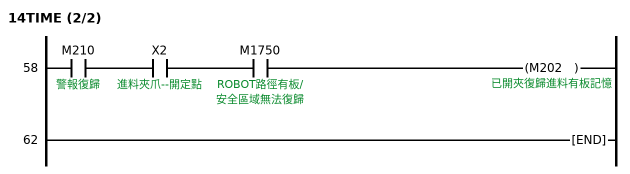
[picture p72: ladder of 14TIME, rungs at steps 58 to 62]
58    LD      M210  ; 警報復歸
      AND     X2  ; 進料夾爪--開定點
      AND     M1750  ; ROBOT路徑有板/安全區域無法復歸
      OUT     M202  ; 已開夾復歸進料有板記憶
62    END
END_PROGRAM

PROGRAM 15STATUS
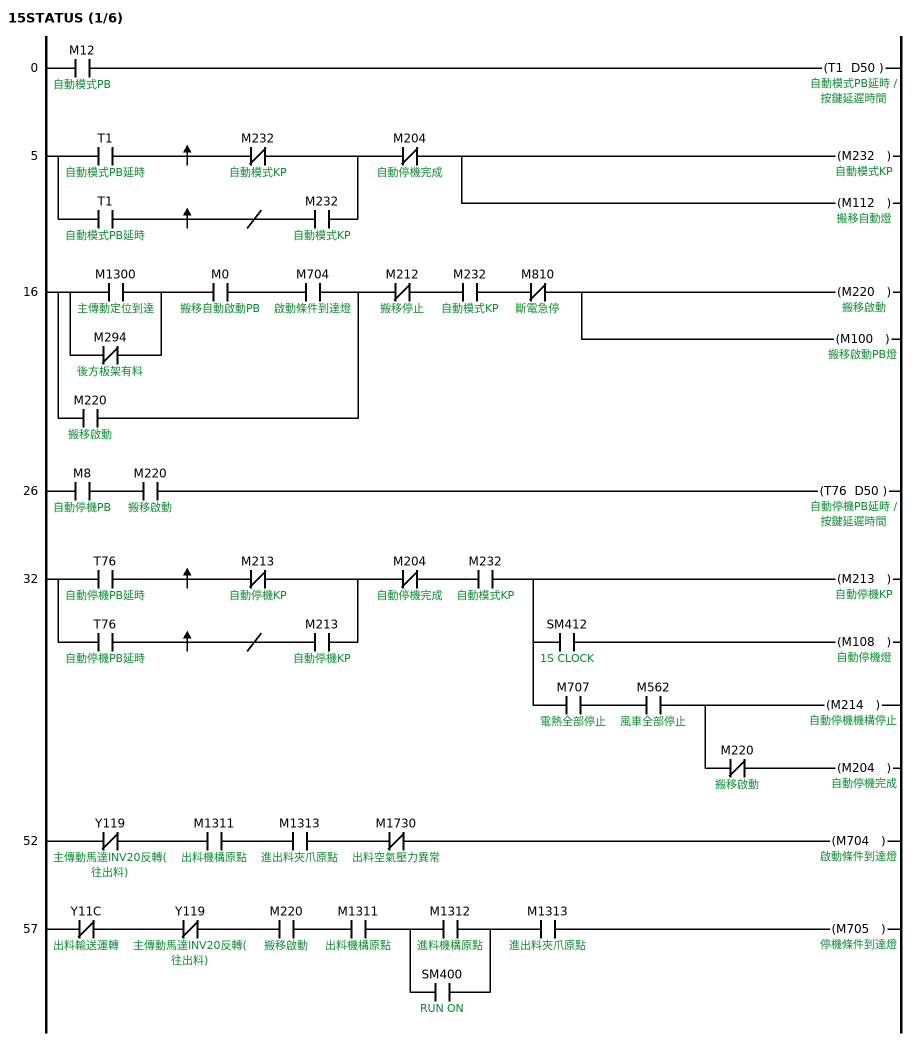
0     LD      M12  ; 自動模式PB
      OUT     T1 D50  ; 自動模式PB延時 / 按鍵延遲時間
5     LD      T1  ; 自動模式PB延時
      MEP
      ANI     M232  ; 自動模式KP
      LD      T1  ; 自動模式PB延時
      MEP
      INV
      AND     M232  ; 自動模式KP
      ORB
      ANI     M204  ; 自動停機完成
      OUT     M232  ; 自動模式KP
      OUT     M112  ; 搬移自動燈
16    LD      M1300  ; 主傳動定位到達
      ORI     M294  ; 後方板架有料
      AND     M0  ; 搬移自動啟動PB
      AND     M704  ; 啟動條件到達燈
      OR      M220  ; 搬移啟動
      ANI     M212  ; 搬移停止
      AND     M232  ; 自動模式KP
      ANI     M810  ; 斷電急停
      OUT     M220  ; 搬移啟動
      OUT     M100  ; 搬移啟動PB燈
26    LD      M8  ; 自動停機PB
      AND     M220  ; 搬移啟動
      OUT     T76 D50  ; 自動停機PB延時 / 按鍵延遲時間
32    LD      T76  ; 自動停機PB延時
      MEP
      ANI     M213  ; 自動停機KP
      LD      T76  ; 自動停機PB延時
      MEP
      INV
      AND     M213  ; 自動停機KP
      ORB
      ANI     M204  ; 自動停機完成
      AND     M232  ; 自動模式KP
      OUT     M213  ; 自動停機KP
      MPS
      AND     SM412  ; 1S CLOCK
      OUT     M108  ; 自動停機燈
      MPP
      AND     M707  ; 電熱全部停止
      AND     M562  ; 風車全部停止
      OUT     M214  ; 自動停機機構停止
      ANI     M220  ; 搬移啟動
      OUT     M204  ; 自動停機完成
52    LDI     Y119  ; 主傳動馬達INV20反轉(往出料)
      AND     M1311  ; 出料機構原點
      AND     M1313  ; 進出料夾爪原點
      ANI     M1730  ; 出料空氣壓力異常
      OUT     M704  ; 啟動條件到達燈
57    LDI     Y11C  ; 出料輸送運轉
      ANI     Y119  ; 主傳動馬達INV20反轉(往出料)
      AND     M220  ; 搬移啟動
      AND     M1311  ; 出料機構原點
      LD      M1312  ; 進料機構原點
      OR      SM400  ; RUN ON
      ANB
      AND     M1313  ; 進出料夾爪原點
      OUT     M705  ; 停機條件到達燈
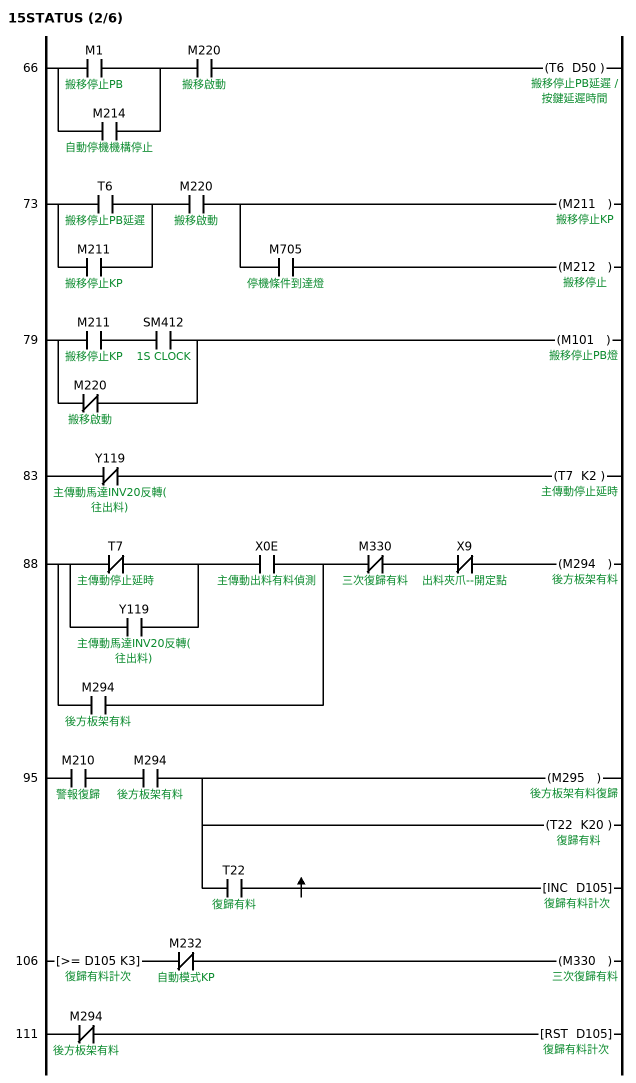
66    LD      M1  ; 搬移停止PB
      OR      M214  ; 自動停機機構停止
      AND     M220  ; 搬移啟動
      OUT     T6 D50  ; 搬移停止PB延遲 / 按鍵延遲時間
73    LD      T6  ; 搬移停止PB延遲
      OR      M211  ; 搬移停止KP
      AND     M220  ; 搬移啟動
      OUT     M211  ; 搬移停止KP
      AND     M705  ; 停機條件到達燈
      OUT     M212  ; 搬移停止
79    LD      M211  ; 搬移停止KP
      AND     SM412  ; 1S CLOCK
      ORI     M220  ; 搬移啟動
      OUT     M101  ; 搬移停止PB燈
83    LDI     Y119  ; 主傳動馬達INV20反轉(往出料)
      OUT     T7 K2  ; 主傳動停止延時
88    LDI     T7  ; 主傳動停止延時
      OR      Y119  ; 主傳動馬達INV20反轉(往出料)
      AND     X0E  ; 主傳動出料有料偵測
      OR      M294  ; 後方板架有料
      ANI     M330  ; 三次復歸有料
      ANI     X9  ; 出料夾爪--開定點
      OUT     M294  ; 後方板架有料
95    LD      M210  ; 警報復歸
      AND     M294  ; 後方板架有料
      OUT     M295  ; 後方板架有料復歸
      OUT     T22 K20  ; 復歸有料
      AND     T22  ; 復歸有料
      MEP
      INC     D105  ; 復歸有料計次
106   LD>=    D105 K3  ; 復歸有料計次
      ANI     M232  ; 自動模式KP
      OUT     M330  ; 三次復歸有料
111   LDI     M294  ; 後方板架有料
      RST     D105  ; 復歸有料計次
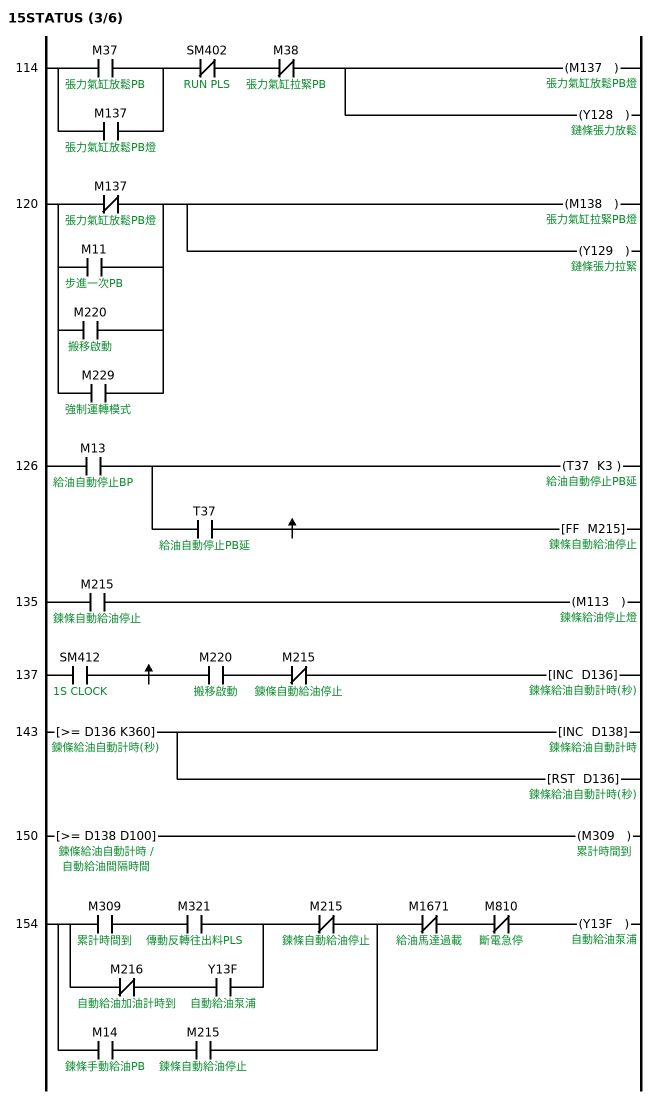
114   LD      M37  ; 張力氣缸放鬆PB
      OR      M137  ; 張力氣缸放鬆PB燈
      ANI     SM402  ; RUN PLS
      ANI     M38  ; 張力氣缸拉緊PB
      OUT     M137  ; 張力氣缸放鬆PB燈
      OUT     Y128  ; 鏈條張力放鬆
120   LDI     M137  ; 張力氣缸放鬆PB燈
      OR      M11  ; 步進一次PB
      OR      M220  ; 搬移啟動
      OR      M229  ; 強制運轉模式
      OUT     M138  ; 張力氣缸拉緊PB燈
      OUT     Y129  ; 鏈條張力拉緊
126   LD      M13  ; 給油自動停止BP
      OUT     T37 K3  ; 給油自動停止PB延
      AND     T37  ; 給油自動停止PB延
      MEP
      FF      M215  ; 鍊條自動給油停止
135   LD      M215  ; 鍊條自動給油停止
      OUT     M113  ; 鍊條給油停止燈
137   LD      SM412  ; 1S CLOCK
      MEP
      AND     M220  ; 搬移啟動
      ANI     M215  ; 鍊條自動給油停止
      INC     D136  ; 鍊條給油自動計時(秒)
143   LD>=    D136 K360  ; 鍊條給油自動計時(秒)
      INC     D138  ; 鍊條給油自動計時
      RST     D136  ; 鍊條給油自動計時(秒)
150   LD>=    D138 D100  ; 鍊條給油自動計時 / 自動給油間隔時間
      OUT     M309  ; 累計時間到
154   LD      M309  ; 累計時間到
      AND     M321  ; 傳動反轉往出料PLS
      LDI     M216  ; 自動給油加油計時到
      AND     Y13F  ; 自動給油泵浦
      ORB
      ANI     M215  ; 鍊條自動給油停止
      LD      M14  ; 鍊條手動給油PB
      AND     M215  ; 鍊條自動給油停止
      ORB
      ANI     M1671  ; 給油馬達過載
      ANI     M810  ; 斷電急停
      OUT     Y13F  ; 自動給油泵浦
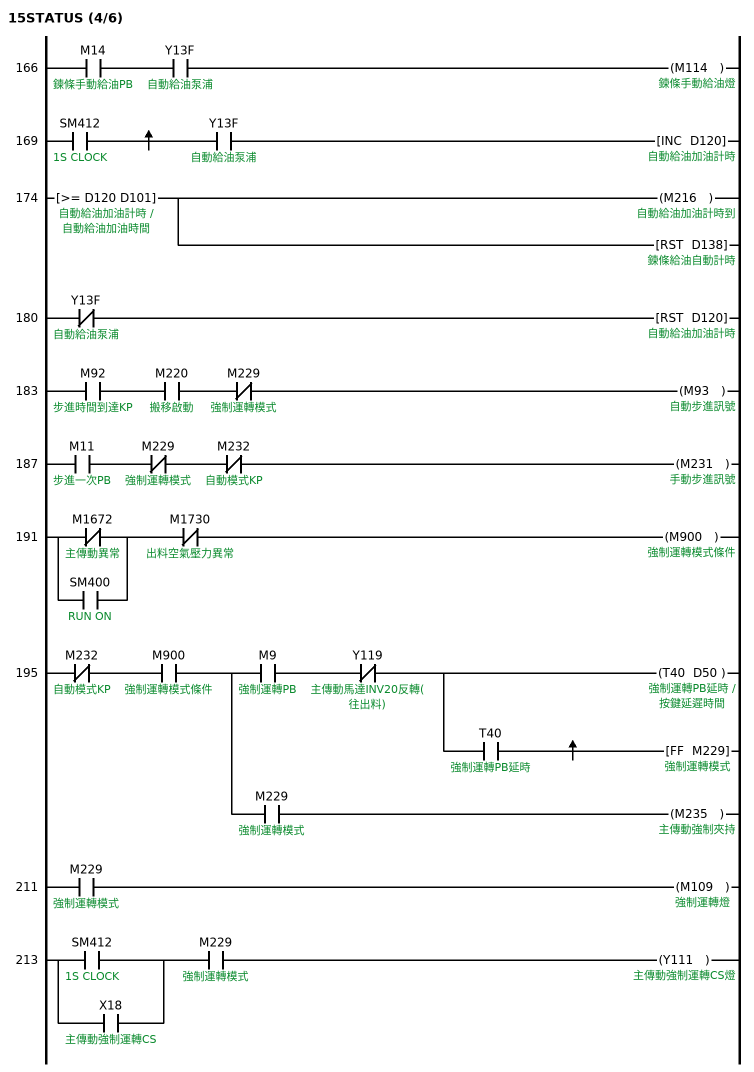
166   LD      M14  ; 鍊條手動給油PB
      AND     Y13F  ; 自動給油泵浦
      OUT     M114  ; 鍊條手動給油燈
169   LD      SM412  ; 1S CLOCK
      MEP
      AND     Y13F  ; 自動給油泵浦
      INC     D120  ; 自動給油加油計時
174   LD>=    D120 D101  ; 自動給油加油計時 / 自動給油加油時間
      OUT     M216  ; 自動給油加油計時到
      RST     D138  ; 鍊條給油自動計時
180   LDI     Y13F  ; 自動給油泵浦
      RST     D120  ; 自動給油加油計時
183   LD      M92  ; 步進時間到達KP
      AND     M220  ; 搬移啟動
      ANI     M229  ; 強制運轉模式
      OUT     M93  ; 自動步進訊號
187   LD      M11  ; 步進一次PB
      ANI     M229  ; 強制運轉模式
      ANI     M232  ; 自動模式KP
      OUT     M231  ; 手動步進訊號
191   LDI     M1672  ; 主傳動異常
      OR      SM400  ; RUN ON
      ANI     M1730  ; 出料空氣壓力異常
      OUT     M900  ; 強制運轉模式條件
195   LDI     M232  ; 自動模式KP
      AND     M900  ; 強制運轉模式條件
      MPS
      AND     M9  ; 強制運轉PB
      ANI     Y119  ; 主傳動馬達INV20反轉(往出料)
      OUT     T40 D50  ; 強制運轉PB延時 / 按鍵延遲時間
      AND     T40  ; 強制運轉PB延時
      MEP
      FF      M229
      MPP
      AND     M229  ; 強制運轉模式
      OUT     M235  ; 主傳動強制夾持
211   LD      M229  ; 強制運轉模式
      OUT     M109  ; 強制運轉燈
213   LD      SM412  ; 1S CLOCK
      OR      X18  ; 主傳動強制運轉CS
      AND     M229  ; 強制運轉模式
      OUT     Y111  ; 主傳動強制運轉CS燈
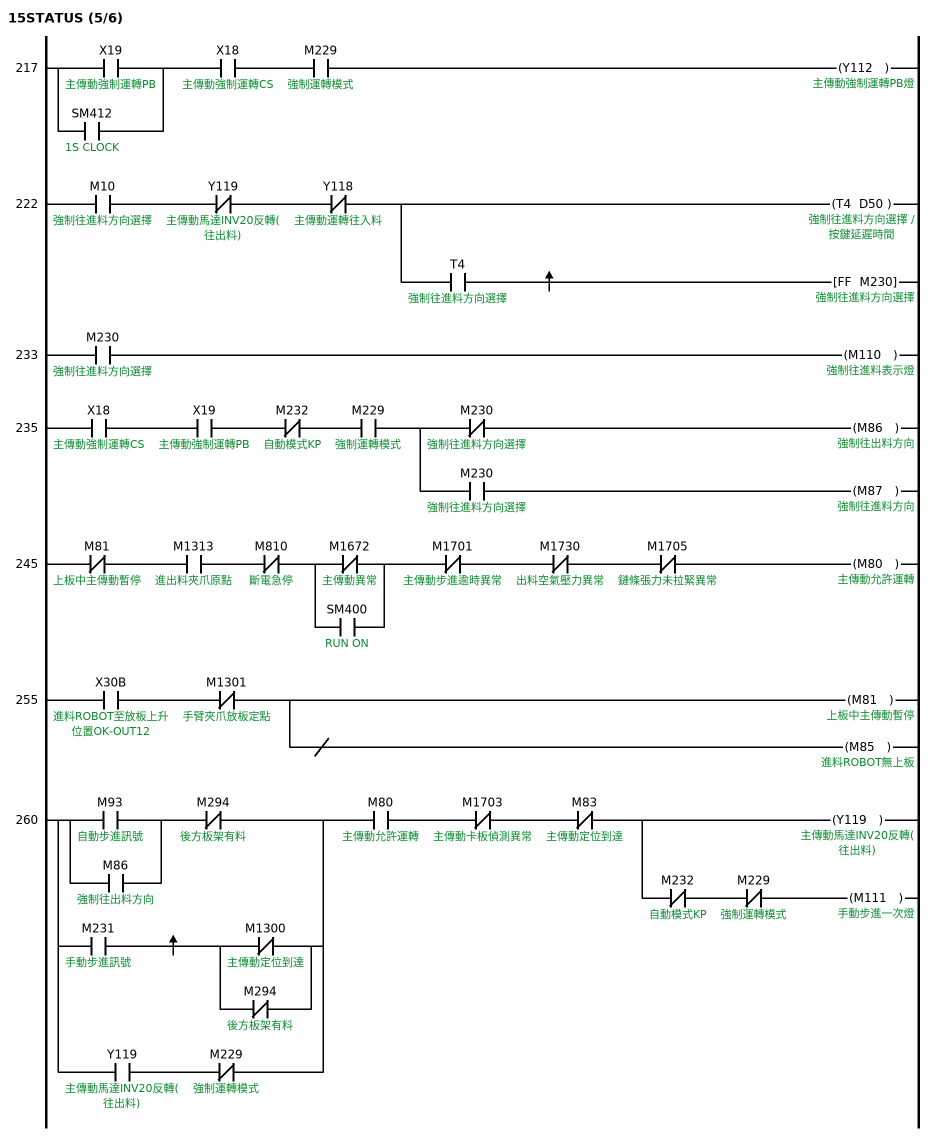
217   LD      X19  ; 主傳動強制運轉PB
      OR      SM412  ; 1S CLOCK
      AND     X18  ; 主傳動強制運轉CS
      AND     M229  ; 強制運轉模式
      OUT     Y112  ; 主傳動強制運轉PB燈
222   LD      M10  ; 強制往進料方向選擇
      ANI     Y119  ; 主傳動馬達INV20反轉(往出料)
      ANI     Y118  ; 主傳動運轉往入料
      OUT     T4 D50  ; 強制往進料方向選擇 / 按鍵延遲時間
      AND     T4  ; 強制往進料方向選擇
      MEP
      FF      M230  ; 強制往進料方向選擇
233   LD      M230  ; 強制往進料方向選擇
      OUT     M110  ; 強制往進料表示燈
235   LD      X18  ; 主傳動強制運轉CS
      AND     X19  ; 主傳動強制運轉PB
      ANI     M232  ; 自動模式KP
      AND     M229  ; 強制運轉模式
      MPS
      ANI     M230  ; 強制往進料方向選擇
      OUT     M86  ; 強制往出料方向
      MPP
      AND     M230  ; 強制往進料方向選擇
      OUT     M87  ; 強制往進料方向
245   LDI     M81  ; 上板中主傳動暫停
      AND     M1313  ; 進出料夾爪原點
      ANI     M810  ; 斷電急停
      LDI     M1672  ; 主傳動異常
      OR      SM400  ; RUN ON
      ANB
      ANI     M1701  ; 主傳動步進逾時異常
      ANI     M1730  ; 出料空氣壓力異常
      ANI     M1705  ; 鏈條張力未拉緊異常
      OUT     M80  ; 主傳動允許運轉
255   LD      X30B  ; 進料ROBOT至放板上升位置OK-OUT12
      ANI     M1301  ; 手臂夾爪放板定點
      OUT     M81  ; 上板中主傳動暫停
      INV
      OUT     M85  ; 進料ROBOT無上板
260   LD      M93  ; 自動步進訊號
      OR      M86  ; 強制往出料方向
      ANI     M294  ; 後方板架有料
      LD      M231  ; 手動步進訊號
      MEP
      LDI     M1300  ; 主傳動定位到達
      ORI     M294  ; 後方板架有料
      ANB
      ORB
      LD      Y119  ; 主傳動馬達INV20反轉(往出料)
      ANI     M229  ; 強制運轉模式
      ORB
      AND     M80  ; 主傳動允許運轉
      ANI     M1703  ; 主傳動卡板偵測異常
      ANI     M83  ; 主傳動定位到達
      OUT     Y119  ; 主傳動馬達INV20反轉(往出料)
      ANI     M232  ; 自動模式KP
      ANI     M229  ; 強制運轉模式
      OUT     M111  ; 手動步進一次燈
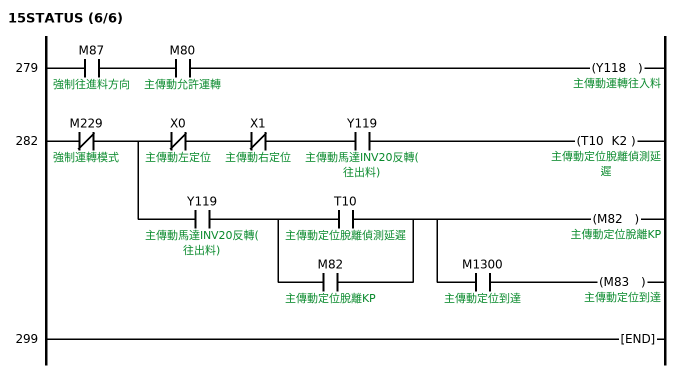
279   LD      M87  ; 強制往進料方向
      AND     M80  ; 主傳動允許運轉
      OUT     Y118  ; 主傳動運轉往入料
282   LDI     M229  ; 強制運轉模式
      MPS
      ANI     X0  ; 主傳動左定位
      ANI     X1  ; 主傳動右定位
      AND     Y119  ; 主傳動馬達INV20反轉(往出料)
      OUT     T10 K2  ; 主傳動定位脫離偵測延遲
      MPP
      AND     Y119  ; 主傳動馬達INV20反轉(往出料)
      LD      T10  ; 主傳動定位脫離偵測延遲
      OR      M82  ; 主傳動定位脫離KP
      ANB
      OUT     M82  ; 主傳動定位脫離KP
      AND     M1300  ; 主傳動定位到達
      OUT     M83  ; 主傳動定位到達
299   END
END_PROGRAM

PROGRAM 21SECS
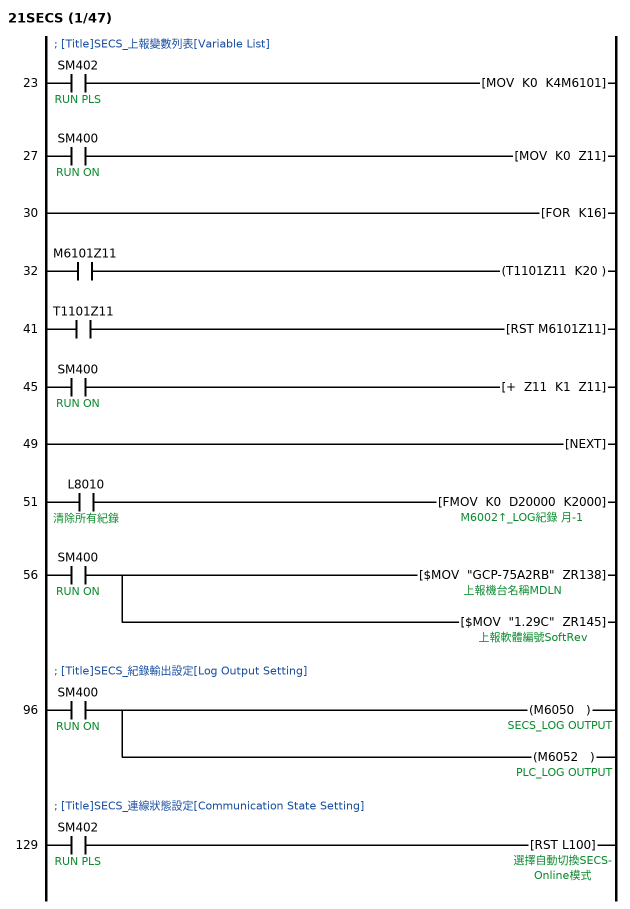
; [Title]SECS_上報變數列表[Variable List]
23    LD      SM402  ; RUN PLS
      MOV     K0 K4M6101  ; EQP->SES控制模式切換(Online/Off)
27    LD      SM400  ; RUN ON
      MOV     K0 Z11
30    FOR     K16
32    LD      M6101Z11
      OUT     T1101Z11 K20
41    LD      T1101Z11
      RST     M6101Z11
45    LD      SM400  ; RUN ON
      +       Z11 K1 Z11
49    NEXT
51    LD      L8010  ; 清除所有紀錄
      FMOV    K0 D20000 K2000  ; M6002↑_LOG紀錄 月-1
56    LD      SM400  ; RUN ON
      $MOV    "GCP-75A2RB" ZR138  ; 上報機台名稱MDLN
      $MOV    "1.29C" ZR145  ; 上報軟體編號SoftRev
; [Title]SECS_紀錄輸出設定[Log Output Setting]
96    LD      SM400  ; RUN ON
      OUT     M6050  ; SECS_LOG OUTPUT
      OUT     M6052  ; PLC_LOG OUTPUT
; [Title]SECS_連線狀態設定[Communication State Setting]
129   LD      SM402  ; RUN PLS
      RST     L100  ; 選擇自動切換SECS-Online模式
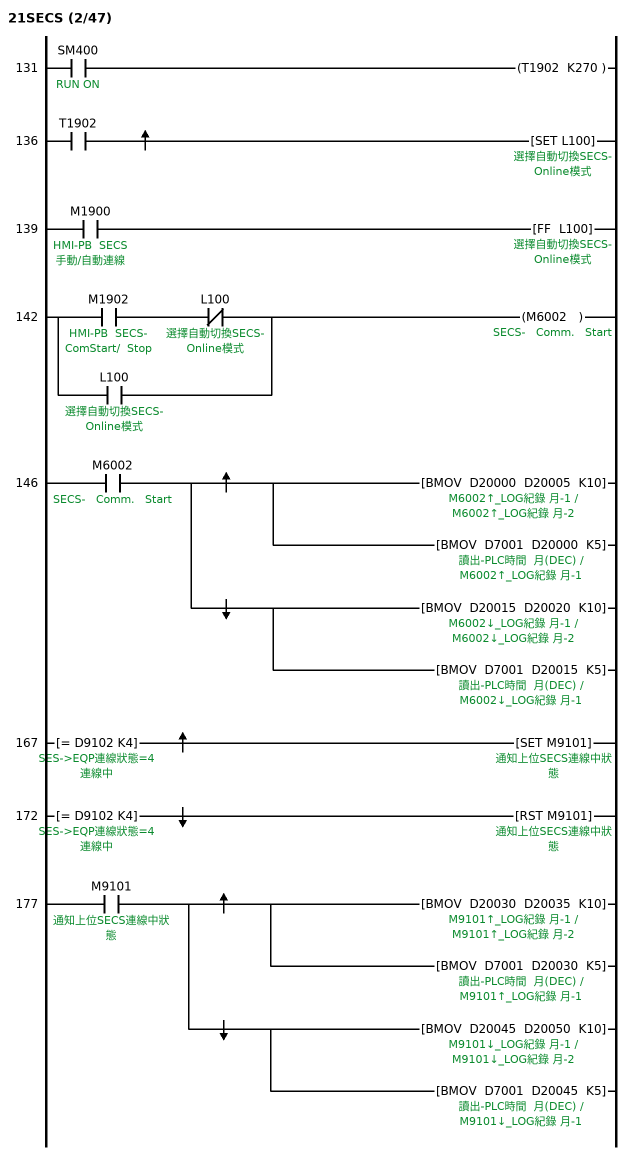
131   LD      SM400  ; RUN ON
      OUT     T1902 K270
136   LD      T1902
      MEP
      SET     L100  ; 選擇自動切換SECS-Online模式
139   LD      M1900  ; HMI-PB  SECS    手動/自動連線
      FF      L100
142   LD      M1902  ; HMI-PB  SECS-ComStart/  Stop
      ANI     L100  ; 選擇自動切換SECS-Online模式
      OR      L100  ; 選擇自動切換SECS-Online模式
      OUT     M6002  ; SECS-   Comm.   Start
146   LD      M6002  ; SECS-   Comm.   Start
      MPS
      MEP
      BMOV    D20000 D20005 K10  ; M6002↑_LOG紀錄 月-2
      BMOV    D7001 D20000 K5  ; 讀出-PLC時間  月(DEC)
      MPP
      MEF
      BMOV    D20015 D20020 K10  ; M6002↓_LOG紀錄 月-1 / M6002↓_LOG紀錄 月-2
      BMOV    D7001 D20015 K5
167   LD=     D9102 K4  ; SES->EQP連線狀態=4      連線中
      MEP
      SET     M9101  ; 通知上位SECS連線中狀態
172   LD=     D9102 K4  ; SES->EQP連線狀態=4      連線中
      MEF
      RST     M9101  ; 通知上位SECS連線中狀態
177   LD      M9101  ; 通知上位SECS連線中狀態
      MPS
      MEP
      BMOV    D20030 D20035 K10  ; M9101↑_LOG紀錄 月-1 / M9101↑_LOG紀錄 月-2
      BMOV    D7001 D20030 K5
      MPP
      MEF
      BMOV    D20045 D20050 K10  ; M9101↓_LOG紀錄 月-1 / M9101↓_LOG紀錄 月-2
      BMOV    D7001 D20045 K5
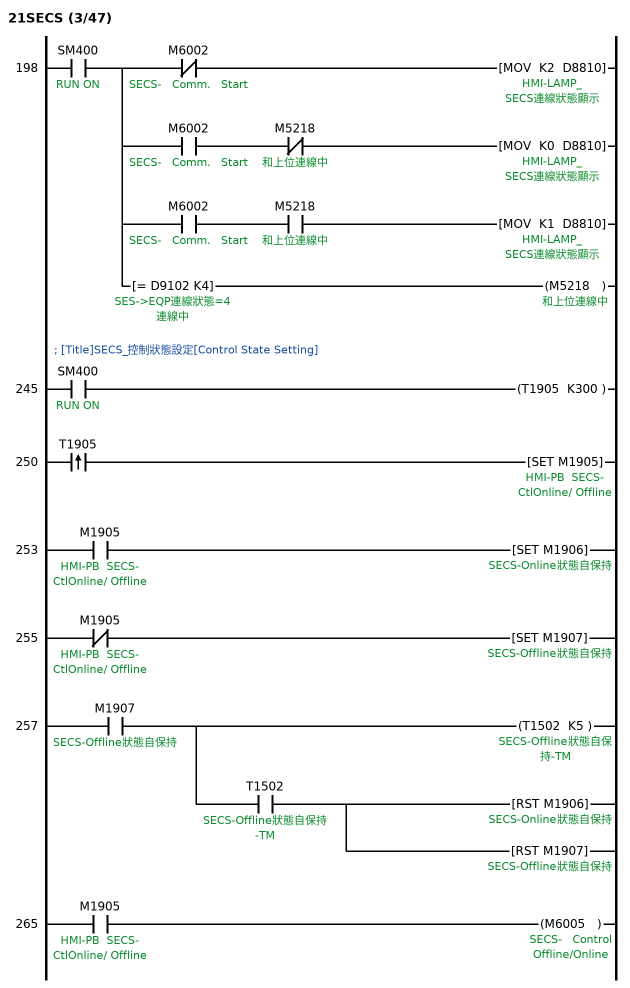
198   LD      SM400  ; RUN ON
      MPS
      ANI     M6002  ; SECS-   Comm.   Start
      MOV     K2 D8810  ; HMI-LAMP_SECS連線狀態顯示
      MRD
      AND     M6002  ; SECS-   Comm.   Start
      ANI     M5218  ; 和上位連線中
      MOV     K0 D8810
      MRD
      AND     M6002  ; SECS-   Comm.   Start
      AND     M5218  ; 和上位連線中
      MOV     K1 D8810
      MPP
      AND=    D9102 K4  ; SES->EQP連線狀態=4      連線中
      OUT     M5218  ; 和上位連線中
; [Title]SECS_控制狀態設定[Control State Setting]
245   LD      SM400  ; RUN ON
      OUT     T1905 K300
250   LDP     T1905
      SET     M1905  ; HMI-PB  SECS-CtlOnline/ Offline
253   LD      M1905  ; HMI-PB  SECS-CtlOnline/ Offline
      SET     M1906  ; SECS-Online狀態自保持
255   LDI     M1905  ; HMI-PB  SECS-CtlOnline/ Offline
      SET     M1907  ; SECS-Offline狀態自保持
257   LD      M1907  ; SECS-Offline狀態自保持
      OUT     T1502 K5  ; SECS-Offline狀態自保持-TM
      AND     T1502  ; SECS-Offline狀態自保持-TM
      RST     M1906  ; SECS-Online狀態自保持
      RST     M1907  ; SECS-Offline狀態自保持
265   LD      M1905  ; HMI-PB  SECS-CtlOnline/ Offline
      OUT     M6005  ; SECS-   Control Offline/Online
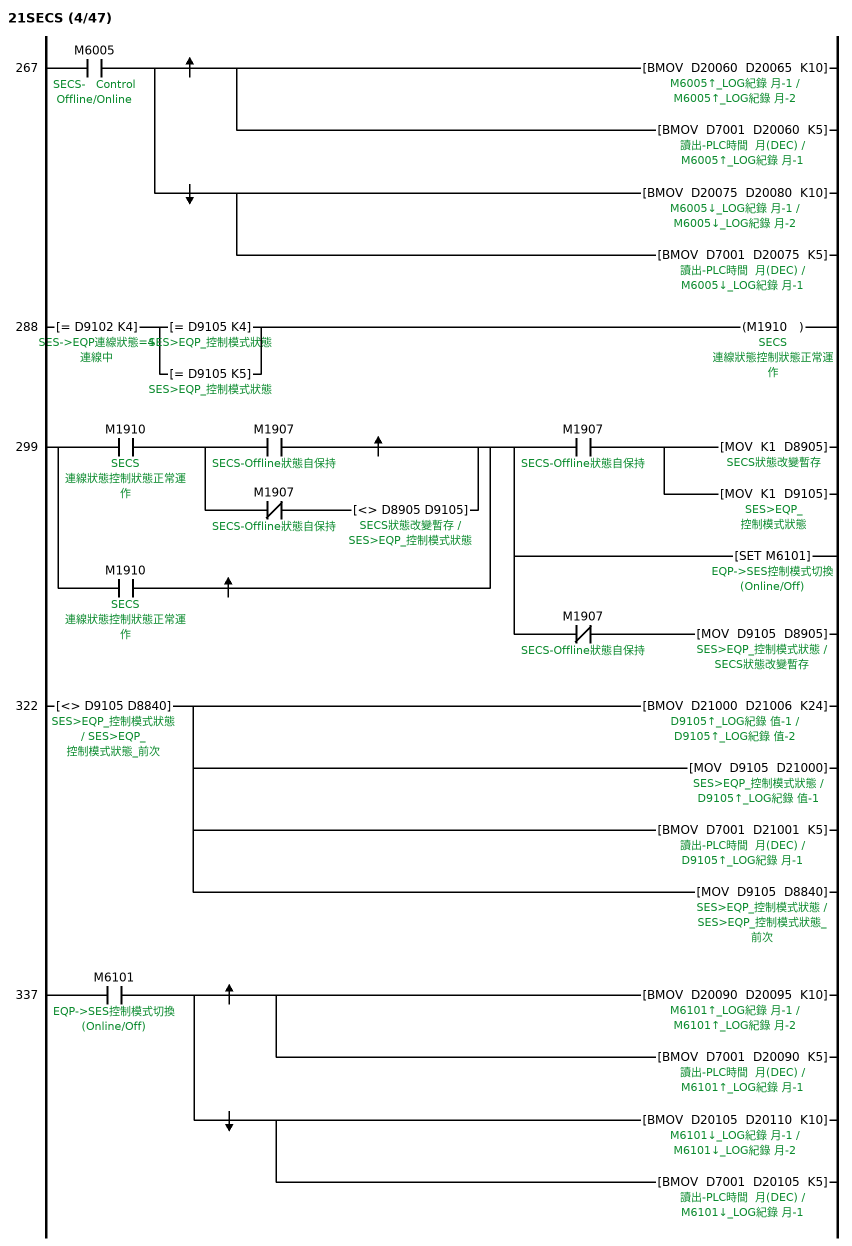
267   LD      M6005  ; SECS-   Control Offline/Online
      MPS
      MEP
      BMOV    D20060 D20065 K10  ; M6005↑_LOG紀錄 月-1 / M6005↑_LOG紀錄 月-2
      BMOV    D7001 D20060 K5
      MPP
      MEF
      BMOV    D20075 D20080 K10  ; M6005↓_LOG紀錄 月-1 / M6005↓_LOG紀錄 月-2
      BMOV    D7001 D20075 K5
288   LD=     D9102 K4  ; SES->EQP連線狀態=4      連線中
      LD=     D9105 K4  ; SES>EQP_控制模式狀態
      OR=     D9105 K5  ; SES>EQP_控制模式狀態
      ANB
      OUT     M1910  ; SECS    連線狀態控制狀態正常運作
299   LD      M1910  ; SECS    連線狀態控制狀態正常運作
      LD      M1907  ; SECS-Offline狀態自保持
      MEP
      LDI     M1907  ; SECS-Offline狀態自保持
      AND<>   D8905 D9105  ; SECS狀態改變暫存 / SES>EQP_控制模式狀態
      ORB
      ANB
      LD      M1910  ; SECS    連線狀態控制狀態正常運作
      MEP
      ORB
      MPS
      AND     M1907  ; SECS-Offline狀態自保持
      MOV     K1 D8905
      MOV     K1 D9105
      MPP
      SET     M6101  ; EQP->SES控制模式切換(Online/Off)
      ANI     M1907  ; SECS-Offline狀態自保持
      MOV     D9105 D8905
322   LD<>    D9105 D8840  ; SES>EQP_控制模式狀態 / SES>EQP_控制模式狀態_前次
      BMOV    D21000 D21006 K24  ; D9105↑_LOG紀錄 值-1 / D9105↑_LOG紀錄 值-2
      MOV     D9105 D21000
      BMOV    D7001 D21001 K5  ; D9105↑_LOG紀錄 月-1
      MOV     D9105 D8840
337   LD      M6101  ; EQP->SES控制模式切換(Online/Off)
      MPS
      MEP
      BMOV    D20090 D20095 K10  ; M6101↑_LOG紀錄 月-1 / M6101↑_LOG紀錄 月-2
      BMOV    D7001 D20090 K5
      MPP
      MEF
      BMOV    D20105 D20110 K10  ; M6101↓_LOG紀錄 月-1 / M6101↓_LOG紀錄 月-2
      BMOV    D7001 D20105 K5
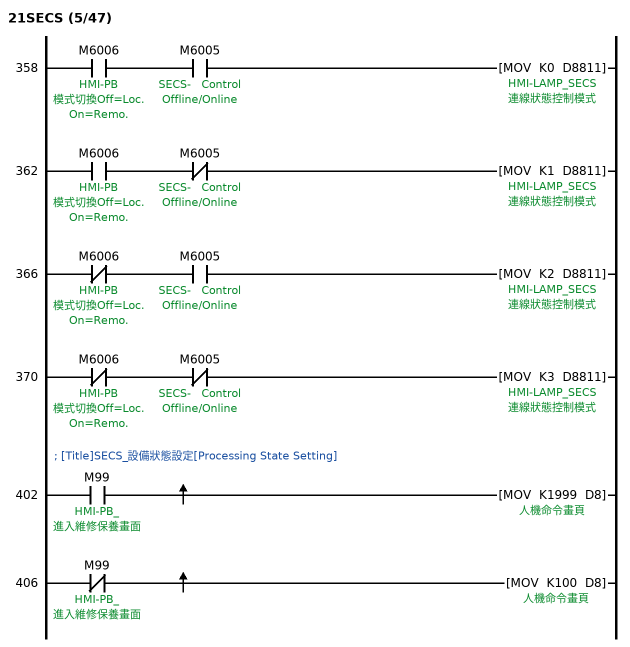
358   LD      M6006  ; HMI-PB  模式切換Off=Loc.On=Remo.
      AND     M6005  ; SECS-   Control Offline/Online
      MOV     K0 D8811  ; HMI-LAMP_SECS   連線狀態控制模式
362   LD      M6006  ; HMI-PB  模式切換Off=Loc.On=Remo.
      ANI     M6005  ; SECS-   Control Offline/Online
      MOV     K1 D8811
366   LDI     M6006  ; HMI-PB  模式切換Off=Loc.On=Remo.
      AND     M6005  ; SECS-   Control Offline/Online
      MOV     K2 D8811
370   LDI     M6006  ; HMI-PB  模式切換Off=Loc.On=Remo.
      ANI     M6005  ; SECS-   Control Offline/Online
      MOV     K3 D8811
; [Title]SECS_設備狀態設定[Processing State Setting]
402   LD      M99  ; HMI-PB_ 進入維修保養畫面
      MEP
      MOV     K1999 D8  ; 人機命令畫頁
406   LDI     M99  ; HMI-PB_ 進入維修保養畫面
      MEP
      MOV     K100 D8
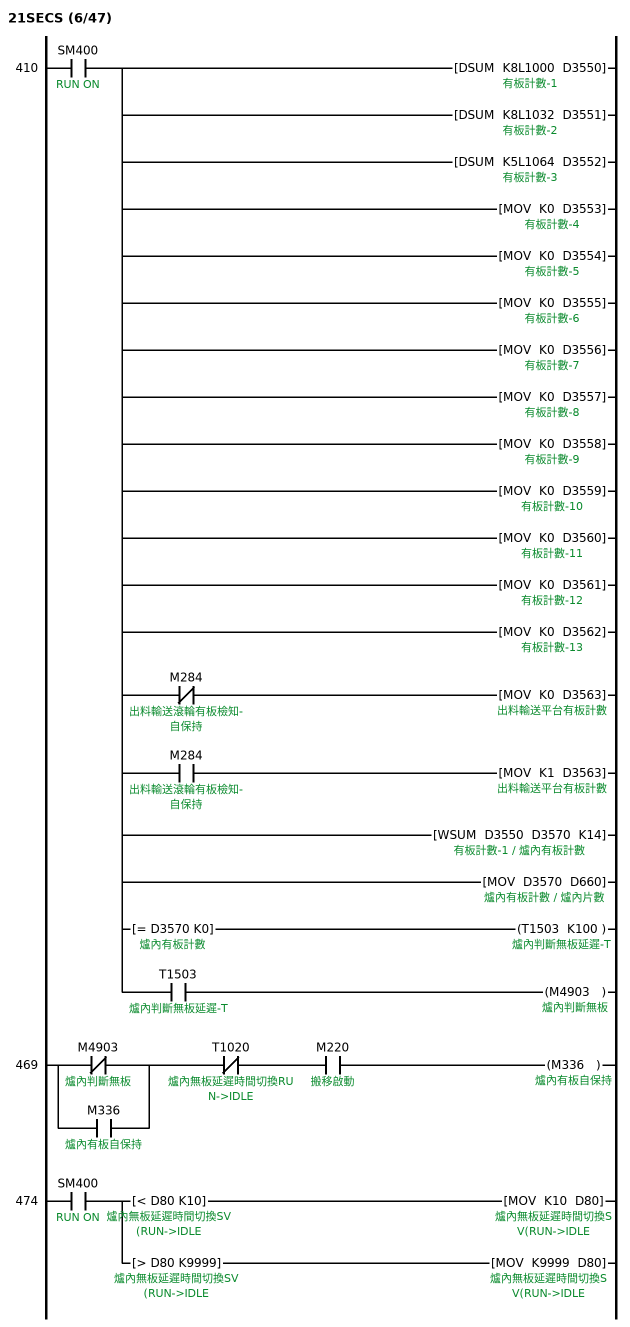
410   LD      SM400  ; RUN ON
      DSUM    K8L1000 D3550  ; 上板記憶 / 有板計數-1
      DSUM    K8L1032 D3551  ; 上板記憶 / 有板計數-2
      DSUM    K5L1064 D3552  ; 上板記憶 / 有板計數-3
      MOV     K0 D3553  ; 有板計數-4
      MOV     K0 D3554  ; 有板計數-5
      MOV     K0 D3555  ; 有板計數-6
      MOV     K0 D3556  ; 有板計數-7
      MOV     K0 D3557  ; 有板計數-8
      MOV     K0 D3558  ; 有板計數-9
      MOV     K0 D3559  ; 有板計數-10
      MOV     K0 D3560  ; 有板計數-11
      MOV     K0 D3561  ; 有板計數-12
      MOV     K0 D3562  ; 有板計數-13
      MPS
      ANI     M284  ; 出料輸送滾輪有板檢知-自保持
      MOV     K0 D3563  ; 出料輸送平台有板計數
      MRD
      AND     M284  ; 出料輸送滾輪有板檢知-自保持
      MOV     K1 D3563
      MPP
      WSUM    D3550 D3570 K14  ; 爐內有板計數
      MOV     D3570 D660  ; 爐內片數
      MPS
      AND=    D3570 K0  ; 爐內有板計數
      OUT     T1503 K100  ; 爐內判斷無板延遲-T
      MPP
      AND     T1503  ; 爐內判斷無板延遲-T
      OUT     M4903  ; 爐內判斷無板
469   LDI     M4903  ; 爐內判斷無板
      OR      M336  ; 爐內有板自保持
      ANI     T1020  ; 爐內無板延遲時間切換RUN->IDLE
      AND     M220  ; 搬移啟動
      OUT     M336  ; 爐內有板自保持
474   LD      SM400  ; RUN ON
      MPS
      AND<    D80 K10  ; 爐內無板延遲時間切換SV(RUN->IDLE
      MOV     K10 D80
      MPP
      AND>    D80 K9999  ; 爐內無板延遲時間切換SV(RUN->IDLE
      MOV     K9999 D80
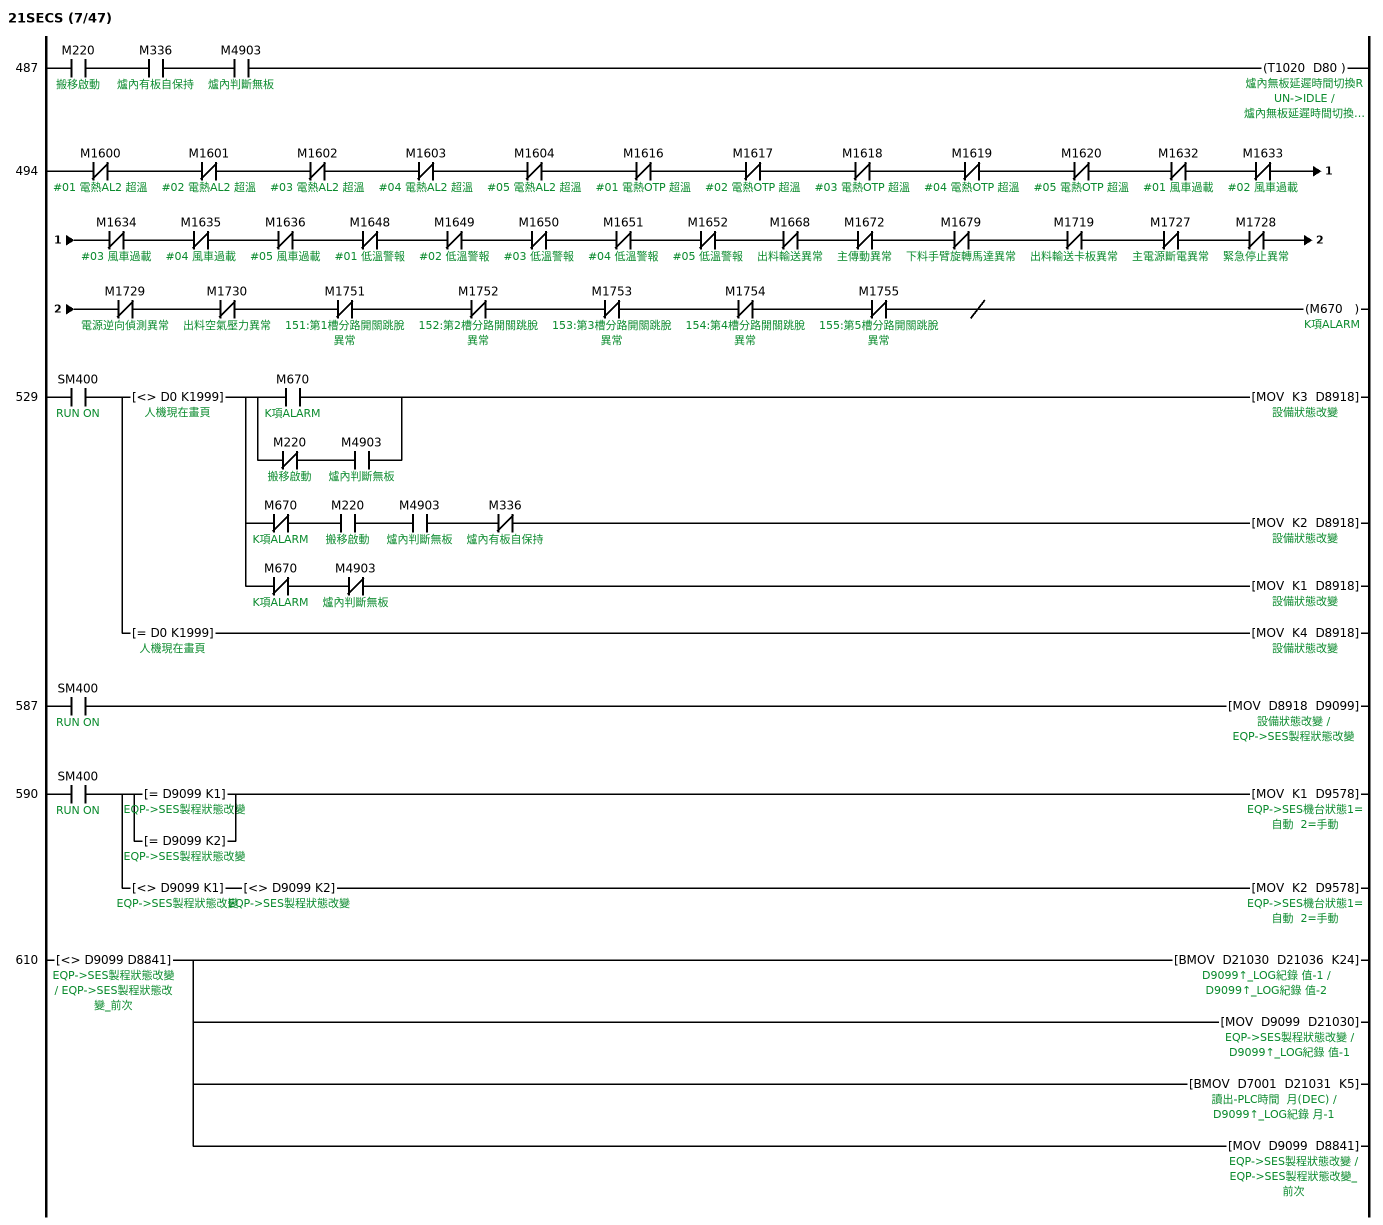
487   LD      M220  ; 搬移啟動
      AND     M336  ; 爐內有板自保持
      AND     M4903  ; 爐內判斷無板
      OUT     T1020 D80  ; 爐內無板延遲時間切換RUN->IDLE / 爐內無板延遲時間切換SV(RUN->IDLE
494   LDI     M1600  ; #01 電熱AL2 超溫
      ANI     M1601  ; #02 電熱AL2 超溫
      ANI     M1602  ; #03 電熱AL2 超溫
      ANI     M1603  ; #04 電熱AL2 超溫
      ANI     M1604  ; #05 電熱AL2 超溫
      ANI     M1616  ; #01 電熱OTP 超溫
      ANI     M1617  ; #02 電熱OTP 超溫
      ANI     M1618  ; #03 電熱OTP 超溫
      ANI     M1619  ; #04 電熱OTP 超溫
      ANI     M1620  ; #05 電熱OTP 超溫
      ANI     M1632  ; #01 風車過載
      ANI     M1633  ; #02 風車過載
      ANI     M1634  ; #03 風車過載
      ANI     M1635  ; #04 風車過載
      ANI     M1636  ; #05 風車過載
      ANI     M1648  ; #01 低溫警報
      ANI     M1649  ; #02 低溫警報
      ANI     M1650  ; #03 低溫警報
      ANI     M1651  ; #04 低溫警報
      ANI     M1652  ; #05 低溫警報
      ANI     M1668  ; 出料輸送異常
      ANI     M1672  ; 主傳動異常
      ANI     M1679  ; 下料手臂旋轉馬達異常
      ANI     M1719  ; 出料輸送卡板異常
      ANI     M1727  ; 主電源斷電異常
      ANI     M1728  ; 緊急停止異常
      ANI     M1729  ; 電源逆向偵測異常
      ANI     M1730  ; 出料空氣壓力異常
      ANI     M1751  ; 151:第1槽分路開關跳脫異常
      ANI     M1752  ; 152:第2槽分路開關跳脫異常
      ANI     M1753  ; 153:第3槽分路開關跳脫異常
      ANI     M1754  ; 154:第4槽分路開關跳脫異常
      ANI     M1755  ; 155:第5槽分路開關跳脫異常
      INV
      OUT     M670  ; K項ALARM
529   LD      SM400  ; RUN ON
      MPS
      AND<>   D0 K1999  ; 人機現在畫頁
      MPS
      LD      M670  ; K項ALARM
      LDI     M220  ; 搬移啟動
      AND     M4903  ; 爐內判斷無板
      ORB
      ANB
      MOV     K3 D8918  ; 設備狀態改變
        [note] State=DOWN
      MRD
      ANI     M670  ; K項ALARM
      AND     M220  ; 搬移啟動
      AND     M4903  ; 爐內判斷無板
      ANI     M336  ; 爐內有板自保持
      MOV     K2 D8918
        [note] State=IDLE
      MPP
      ANI     M670  ; K項ALARM
      ANI     M4903  ; 爐內判斷無板
      MOV     K1 D8918
        [note] State=RUN
      MPP
      AND=    D0 K1999  ; 人機現在畫頁
      MOV     K4 D8918
        [note] State=PM
587   LD      SM400  ; RUN ON
      MOV     D8918 D9099  ; EQP->SES製程狀態改變
590   LD      SM400  ; RUN ON
      MPS
      LD=     D9099 K1  ; EQP->SES製程狀態改變
      OR=     D9099 K2  ; EQP->SES製程狀態改變
      ANB
      MOV     K1 D9578  ; EQP->SES機台狀態1=自動  2=手動
      MPP
      AND<>   D9099 K1  ; EQP->SES製程狀態改變
      AND<>   D9099 K2  ; EQP->SES製程狀態改變
      MOV     K2 D9578
610   LD<>    D9099 D8841  ; EQP->SES製程狀態改變 / EQP->SES製程狀態改變_前次
      BMOV    D21030 D21036 K24  ; D9099↑_LOG紀錄 值-1 / D9099↑_LOG紀錄 值-2
      MOV     D9099 D21030
      BMOV    D7001 D21031 K5  ; D9099↑_LOG紀錄 月-1
      MOV     D9099 D8841
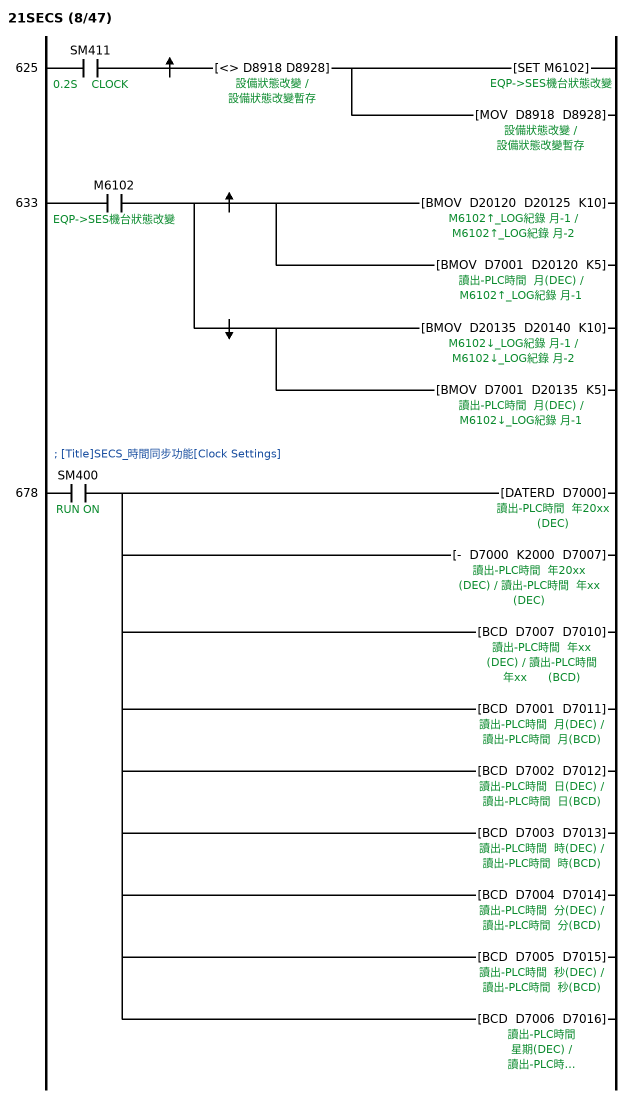
625   LD      SM411  ; 0.2S    CLOCK
      MEP
      AND<>   D8918 D8928  ; 設備狀態改變 / 設備狀態改變暫存
      SET     M6102  ; EQP->SES機台狀態改變
      MOV     D8918 D8928
633   LD      M6102  ; EQP->SES機台狀態改變
      MPS
      MEP
      BMOV    D20120 D20125 K10  ; M6102↑_LOG紀錄 月-1 / M6102↑_LOG紀錄 月-2
      BMOV    D7001 D20120 K5
      MPP
      MEF
      BMOV    D20135 D20140 K10  ; M6102↓_LOG紀錄 月-1 / M6102↓_LOG紀錄 月-2
      BMOV    D7001 D20135 K5
; [Title]SECS_時間同步功能[Clock Settings]
678   LD      SM400  ; RUN ON
      DATERD  D7000  ; 讀出-PLC時間  年20xx    (DEC)
      -       D7000 K2000 D7007  ; 讀出-PLC時間  年xx      (DEC)
      BCD     D7007 D7010  ; 讀出-PLC時間  年xx      (BCD)
      BCD     D7001 D7011  ; 讀出-PLC時間  月(BCD)
      BCD     D7002 D7012  ; 讀出-PLC時間  日(DEC) / 讀出-PLC時間  日(BCD)
      BCD     D7003 D7013  ; 讀出-PLC時間  時(DEC) / 讀出-PLC時間  時(BCD)
      BCD     D7004 D7014  ; 讀出-PLC時間  分(DEC) / 讀出-PLC時間  分(BCD)
      BCD     D7005 D7015  ; 讀出-PLC時間  秒(DEC) / 讀出-PLC時間  秒(BCD)
      BCD     D7006 D7016  ; 讀出-PLC時間  星期(DEC) / 讀出-PLC時間  星期(BCD)
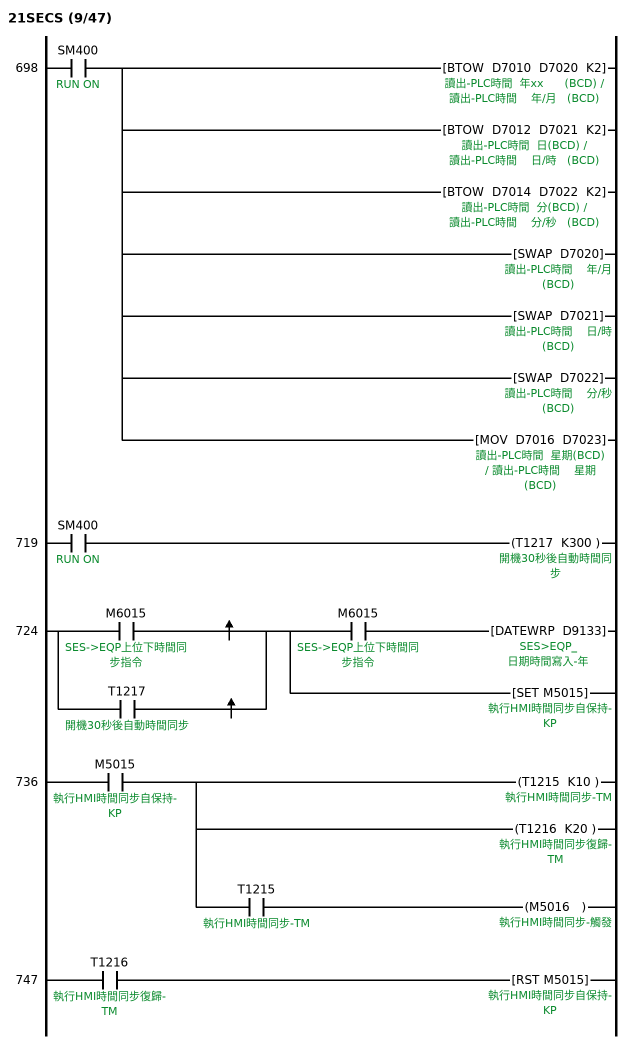
698   LD      SM400  ; RUN ON
      BTOW    D7010 D7020 K2  ; 讀出-PLC時間    年/月   (BCD)
      BTOW    D7012 D7021 K2  ; 讀出-PLC時間    日/時   (BCD)
      BTOW    D7014 D7022 K2  ; 讀出-PLC時間    分/秒   (BCD)
      SWAP    D7020
      SWAP    D7021
      SWAP    D7022
      MOV     D7016 D7023  ; 讀出-PLC時間    星期    (BCD)
719   LD      SM400  ; RUN ON
      OUT     T1217 K300  ; 開機30秒後自動時間同步
724   LD      M6015  ; SES->EQP上位下時間同步指令
      MEP
      LD      T1217  ; 開機30秒後自動時間同步
      MEP
      ORB
      MPS
      AND     M6015  ; SES->EQP上位下時間同步指令
      DATEWRP D9133  ; SES>EQP_日期時間寫入-年
      MPP
      SET     M5015  ; 執行HMI時間同步自保持-KP
736   LD      M5015  ; 執行HMI時間同步自保持-KP
      OUT     T1215 K10  ; 執行HMI時間同步-TM
      OUT     T1216 K20  ; 執行HMI時間同步復歸-TM
      AND     T1215  ; 執行HMI時間同步-TM
      OUT     M5016  ; 執行HMI時間同步-觸發
747   LD      T1216  ; 執行HMI時間同步復歸-TM
      RST     M5015  ; 執行HMI時間同步自保持-KP
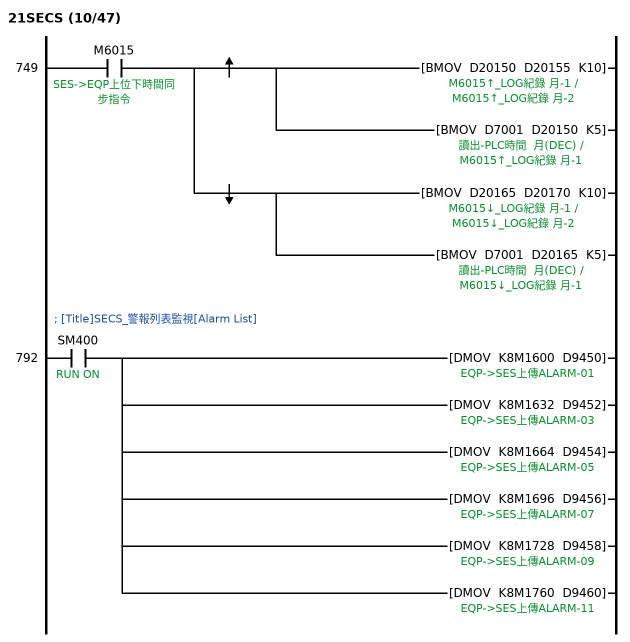
749   LD      M6015  ; SES->EQP上位下時間同步指令
      MPS
      MEP
      BMOV    D20150 D20155 K10  ; M6015↑_LOG紀錄 月-1 / M6015↑_LOG紀錄 月-2
      BMOV    D7001 D20150 K5
      MPP
      MEF
      BMOV    D20165 D20170 K10  ; M6015↓_LOG紀錄 月-1 / M6015↓_LOG紀錄 月-2
      BMOV    D7001 D20165 K5
; [Title]SECS_警報列表監視[Alarm List]
792   LD      SM400  ; RUN ON
      DMOV    K8M1600 D9450  ; EQP->SES上傳ALARM-01
      DMOV    K8M1632 D9452  ; EQP->SES上傳ALARM-03
      DMOV    K8M1664 D9454  ; 進料風車過載異常 / EQP->SES上傳ALARM-05
      DMOV    K8M1696 D9456  ; 進料夾爪開異常 / EQP->SES上傳ALARM-07
      DMOV    K8M1728 D9458  ; EQP->SES上傳ALARM-09
      DMOV    K8M1760 D9460  ; EQP->SES上傳ALARM-11
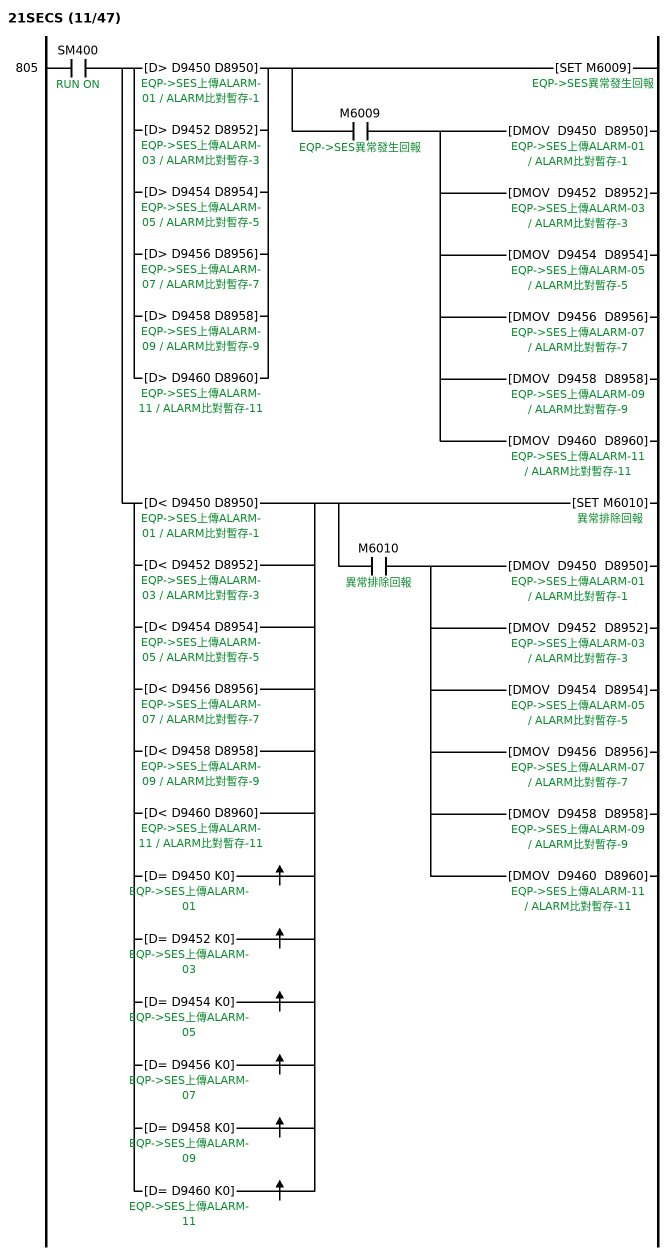
805   LD      SM400  ; RUN ON
      MPS
      LDD>    D9450 D8950  ; EQP->SES上傳ALARM-01 / ALARM比對暫存-1
      ORD>    D9452 D8952  ; EQP->SES上傳ALARM-03 / ALARM比對暫存-3
      ORD>    D9454 D8954  ; EQP->SES上傳ALARM-05 / ALARM比對暫存-5
      ORD>    D9456 D8956  ; EQP->SES上傳ALARM-07 / ALARM比對暫存-7
      ORD>    D9458 D8958  ; EQP->SES上傳ALARM-09 / ALARM比對暫存-9
      ORD>    D9460 D8960  ; EQP->SES上傳ALARM-11 / ALARM比對暫存-11
      ANB
      SET     M6009  ; EQP->SES異常發生回報
      AND     M6009  ; EQP->SES異常發生回報
      DMOV    D9450 D8950
      DMOV    D9452 D8952
      DMOV    D9454 D8954
      DMOV    D9456 D8956
      DMOV    D9458 D8958
      DMOV    D9460 D8960
      MPP
      LDD<    D9450 D8950  ; EQP->SES上傳ALARM-01 / ALARM比對暫存-1
      ORD<    D9452 D8952  ; EQP->SES上傳ALARM-03 / ALARM比對暫存-3
      ORD<    D9454 D8954  ; EQP->SES上傳ALARM-05 / ALARM比對暫存-5
      ORD<    D9456 D8956  ; EQP->SES上傳ALARM-07 / ALARM比對暫存-7
      ORD<    D9458 D8958  ; EQP->SES上傳ALARM-09 / ALARM比對暫存-9
      ORD<    D9460 D8960  ; EQP->SES上傳ALARM-11 / ALARM比對暫存-11
      LDD=    D9450 K0  ; EQP->SES上傳ALARM-01
      MEP
      ORB
      LDD=    D9452 K0  ; EQP->SES上傳ALARM-03
      MEP
      ORB
      LDD=    D9454 K0  ; EQP->SES上傳ALARM-05
      MEP
      ORB
      LDD=    D9456 K0  ; EQP->SES上傳ALARM-07
      MEP
      ORB
      LDD=    D9458 K0  ; EQP->SES上傳ALARM-09
      MEP
      ORB
      LDD=    D9460 K0  ; EQP->SES上傳ALARM-11
      MEP
      ORB
      ANB
      SET     M6010  ; 異常排除回報
      AND     M6010  ; 異常排除回報
      DMOV    D9450 D8950
      DMOV    D9452 D8952
      DMOV    D9454 D8954
      DMOV    D9456 D8956
      DMOV    D9458 D8958
      DMOV    D9460 D8960
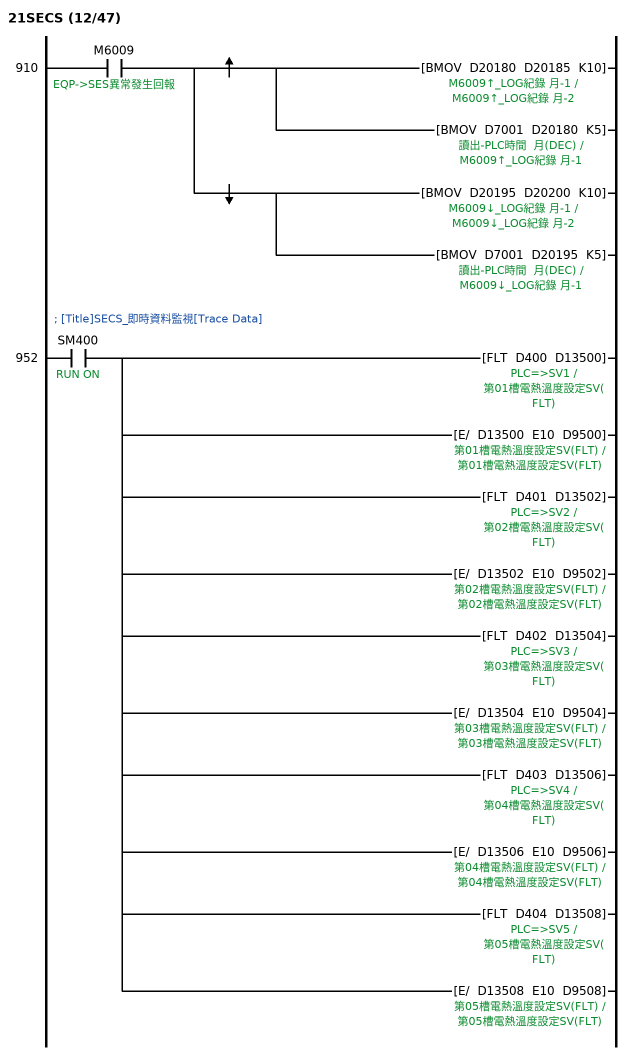
910   LD      M6009  ; EQP->SES異常發生回報
      MPS
      MEP
      BMOV    D20180 D20185 K10  ; M6009↑_LOG紀錄 月-1 / M6009↑_LOG紀錄 月-2
      BMOV    D7001 D20180 K5
      MPP
      MEF
      BMOV    D20195 D20200 K10  ; M6009↓_LOG紀錄 月-1 / M6009↓_LOG紀錄 月-2
      BMOV    D7001 D20195 K5
; [Title]SECS_即時資料監視[Trace Data]
952   LD      SM400  ; RUN ON
      FLT     D400 D13500  ; PLC=>SV1 / 第01槽電熱溫度設定SV(FLT)
      E/      D13500 E10 D9500  ; 第01槽電熱溫度設定SV(FLT)
      FLT     D401 D13502  ; PLC=>SV2 / 第02槽電熱溫度設定SV(FLT)
      E/      D13502 E10 D9502  ; 第02槽電熱溫度設定SV(FLT)
      FLT     D402 D13504  ; PLC=>SV3 / 第03槽電熱溫度設定SV(FLT)
      E/      D13504 E10 D9504  ; 第03槽電熱溫度設定SV(FLT)
      FLT     D403 D13506  ; PLC=>SV4 / 第04槽電熱溫度設定SV(FLT)
      E/      D13506 E10 D9506  ; 第04槽電熱溫度設定SV(FLT)
      FLT     D404 D13508  ; PLC=>SV5 / 第05槽電熱溫度設定SV(FLT)
      E/      D13508 E10 D9508  ; 第05槽電熱溫度設定SV(FLT)
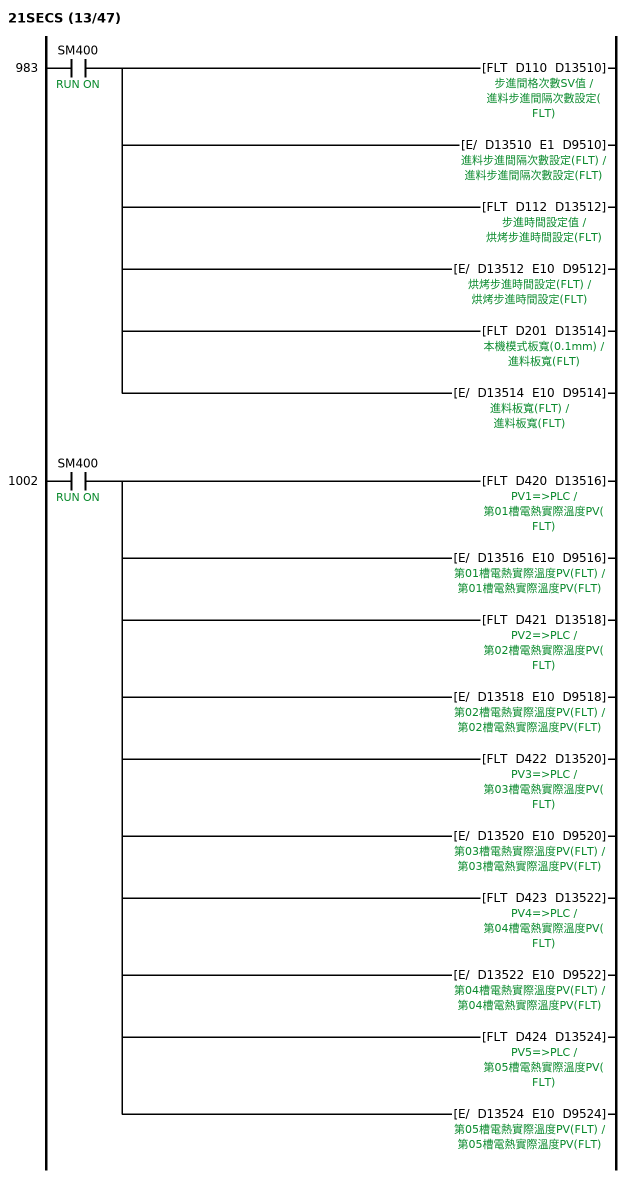
983   LD      SM400  ; RUN ON
      FLT     D110 D13510  ; 步進間格次數SV值 / 進料步進間隔次數設定(FLT)
      E/      D13510 E1 D9510  ; 進料步進間隔次數設定(FLT)
      FLT     D112 D13512  ; 步進時間設定值 / 烘烤步進時間設定(FLT)
      E/      D13512 E10 D9512  ; 烘烤步進時間設定(FLT)
      FLT     D201 D13514  ; 本機模式板寬(0.1mm) / 進料板寬(FLT)
      E/      D13514 E10 D9514  ; 進料板寬(FLT)
1002  LD      SM400  ; RUN ON
      FLT     D420 D13516  ; PV1=>PLC / 第01槽電熱實際溫度PV(FLT)
      E/      D13516 E10 D9516  ; 第01槽電熱實際溫度PV(FLT)
      FLT     D421 D13518  ; PV2=>PLC / 第02槽電熱實際溫度PV(FLT)
      E/      D13518 E10 D9518  ; 第02槽電熱實際溫度PV(FLT)
      FLT     D422 D13520  ; PV3=>PLC / 第03槽電熱實際溫度PV(FLT)
      E/      D13520 E10 D9520  ; 第03槽電熱實際溫度PV(FLT)
      FLT     D423 D13522  ; PV4=>PLC / 第04槽電熱實際溫度PV(FLT)
      E/      D13522 E10 D9522  ; 第04槽電熱實際溫度PV(FLT)
      FLT     D424 D13524  ; PV5=>PLC / 第05槽電熱實際溫度PV(FLT)
      E/      D13524 E10 D9524  ; 第05槽電熱實際溫度PV(FLT)
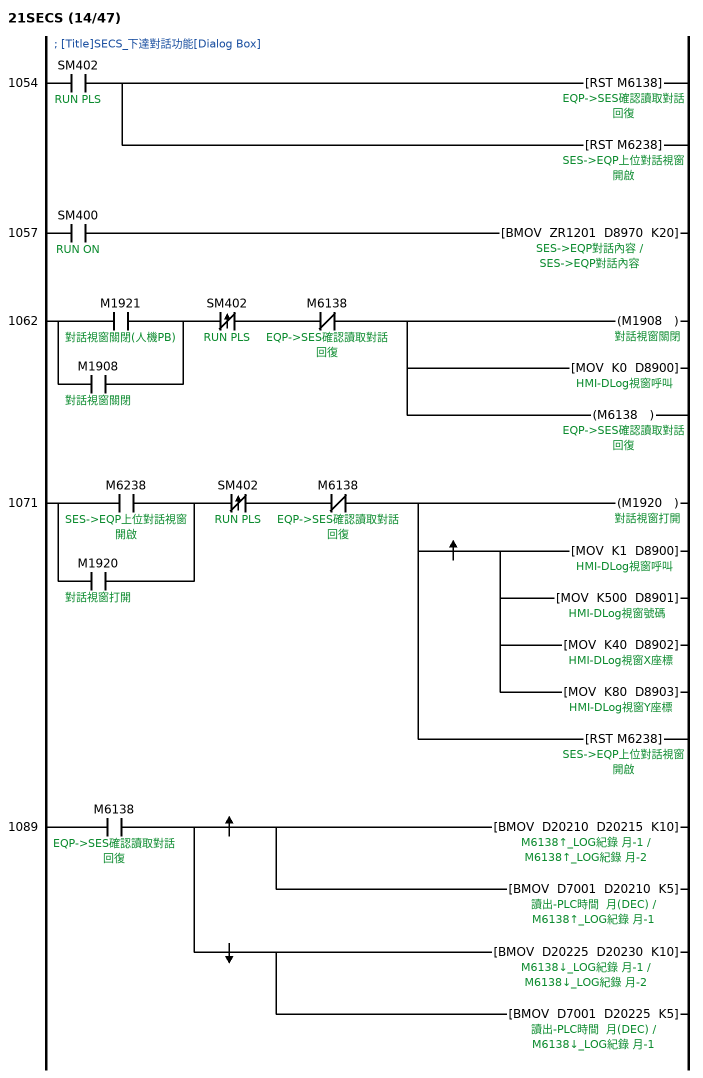
; [Title]SECS_下達對話功能[Dialog Box]
1054  LD      SM402  ; RUN PLS
      RST     M6138  ; EQP->SES確認讀取對話回復
      RST     M6238  ; SES->EQP上位對話視窗開啟
1057  LD      SM400  ; RUN ON
      BMOV    ZR1201 D8970 K20  ; SES->EQP對話內容 / SES->EQP對話內容
1062  LD      M1921  ; 對話視窗關閉(人機PB)
      OR      M1908  ; 對話視窗關閉
      ANDPI   SM402  ; RUN PLS
      ANI     M6138  ; EQP->SES確認讀取對話回復
      OUT     M1908  ; 對話視窗關閉
      MOV     K0 D8900  ; HMI-DLog視窗呼叫
      OUT     M6138  ; EQP->SES確認讀取對話回復
1071  LD      M6238  ; SES->EQP上位對話視窗開啟
      OR      M1920  ; 對話視窗打開
      ANDPI   SM402  ; RUN PLS
      ANI     M6138  ; EQP->SES確認讀取對話回復
      OUT     M1920  ; 對話視窗打開
      MPS
      MEP
      MOV     K1 D8900
      MOV     K500 D8901  ; HMI-DLog視窗號碼
      MOV     K40 D8902  ; HMI-DLog視窗X座標
      MOV     K80 D8903  ; HMI-DLog視窗Y座標
      MPP
      RST     M6238  ; SES->EQP上位對話視窗開啟
1089  LD      M6138  ; EQP->SES確認讀取對話回復
      MPS
      MEP
      BMOV    D20210 D20215 K10  ; M6138↑_LOG紀錄 月-1 / M6138↑_LOG紀錄 月-2
      BMOV    D7001 D20210 K5
      MPP
      MEF
      BMOV    D20225 D20230 K10  ; M6138↓_LOG紀錄 月-1 / M6138↓_LOG紀錄 月-2
      BMOV    D7001 D20225 K5
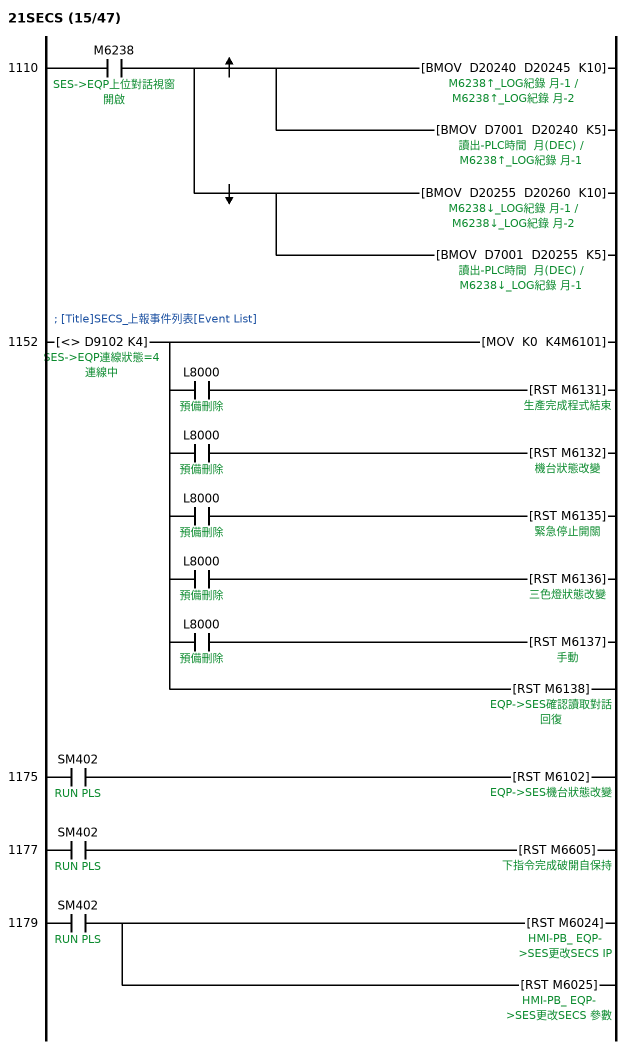
1110  LD      M6238  ; SES->EQP上位對話視窗開啟
      MPS
      MEP
      BMOV    D20240 D20245 K10  ; M6238↑_LOG紀錄 月-1 / M6238↑_LOG紀錄 月-2
      BMOV    D7001 D20240 K5
      MPP
      MEF
      BMOV    D20255 D20260 K10  ; M6238↓_LOG紀錄 月-1 / M6238↓_LOG紀錄 月-2
      BMOV    D7001 D20255 K5
; [Title]SECS_上報事件列表[Event List]
1152  LD<>    D9102 K4  ; SES->EQP連線狀態=4      連線中
      MOV     K0 K4M6101
      MPS
      AND     L8000  ; 預備刪除
      RST     M6131  ; 生產完成程式結束
      MRD
      AND     L8000  ; 預備刪除
      RST     M6132  ; 機台狀態改變
      MRD
      AND     L8000  ; 預備刪除
      RST     M6135  ; 緊急停止開關
      MRD
      AND     L8000  ; 預備刪除
      RST     M6136  ; 三色燈狀態改變
      MRD
      AND     L8000  ; 預備刪除
      RST     M6137  ; 手動
      MPP
      RST     M6138  ; EQP->SES確認讀取對話回復
1175  LD      SM402  ; RUN PLS
      RST     M6102  ; EQP->SES機台狀態改變
1177  LD      SM402  ; RUN PLS
      RST     M6605  ; 下指令完成破開自保持
1179  LD      SM402  ; RUN PLS
      RST     M6024  ; HMI-PB_ EQP->SES更改SECS IP
        [note] HMI上變更C語言模組網路設定
      RST     M6025  ; HMI-PB_ EQP->SES更改SECS 參數
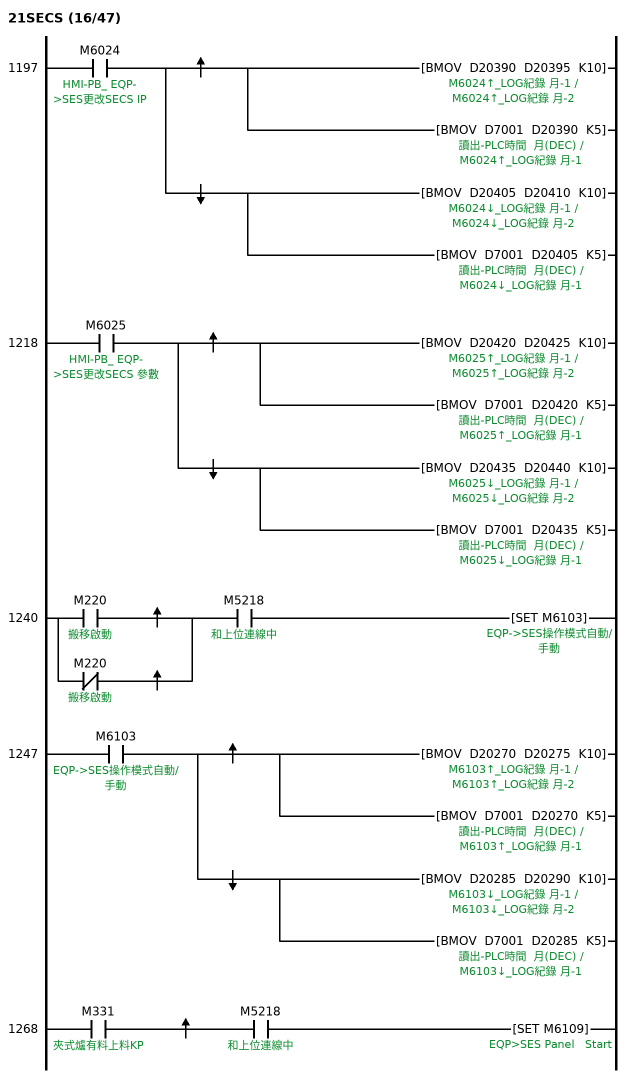
1197  LD      M6024  ; HMI-PB_ EQP->SES更改SECS IP
      MPS
      MEP
      BMOV    D20390 D20395 K10  ; M6024↑_LOG紀錄 月-1 / M6024↑_LOG紀錄 月-2
      BMOV    D7001 D20390 K5
      MPP
      MEF
      BMOV    D20405 D20410 K10  ; M6024↓_LOG紀錄 月-1 / M6024↓_LOG紀錄 月-2
      BMOV    D7001 D20405 K5
1218  LD      M6025  ; HMI-PB_ EQP->SES更改SECS 參數
      MPS
      MEP
      BMOV    D20420 D20425 K10  ; M6025↑_LOG紀錄 月-1 / M6025↑_LOG紀錄 月-2
      BMOV    D7001 D20420 K5
      MPP
      MEF
      BMOV    D20435 D20440 K10  ; M6025↓_LOG紀錄 月-1 / M6025↓_LOG紀錄 月-2
      BMOV    D7001 D20435 K5
1240  LD      M220  ; 搬移啟動
      MEP
      LDI     M220  ; 搬移啟動
      MEP
      ORB
      AND     M5218  ; 和上位連線中
      SET     M6103  ; EQP->SES操作模式自動/手動
1247  LD      M6103  ; EQP->SES操作模式自動/手動
      MPS
      MEP
      BMOV    D20270 D20275 K10  ; M6103↑_LOG紀錄 月-1 / M6103↑_LOG紀錄 月-2
      BMOV    D7001 D20270 K5
      MPP
      MEF
      BMOV    D20285 D20290 K10  ; M6103↓_LOG紀錄 月-1 / M6103↓_LOG紀錄 月-2
      BMOV    D7001 D20285 K5
1268  LD      M331  ; 夾式爐有料上料KP
      MEP
      AND     M5218  ; 和上位連線中
      SET     M6109  ; EQP>SES Panel   Start
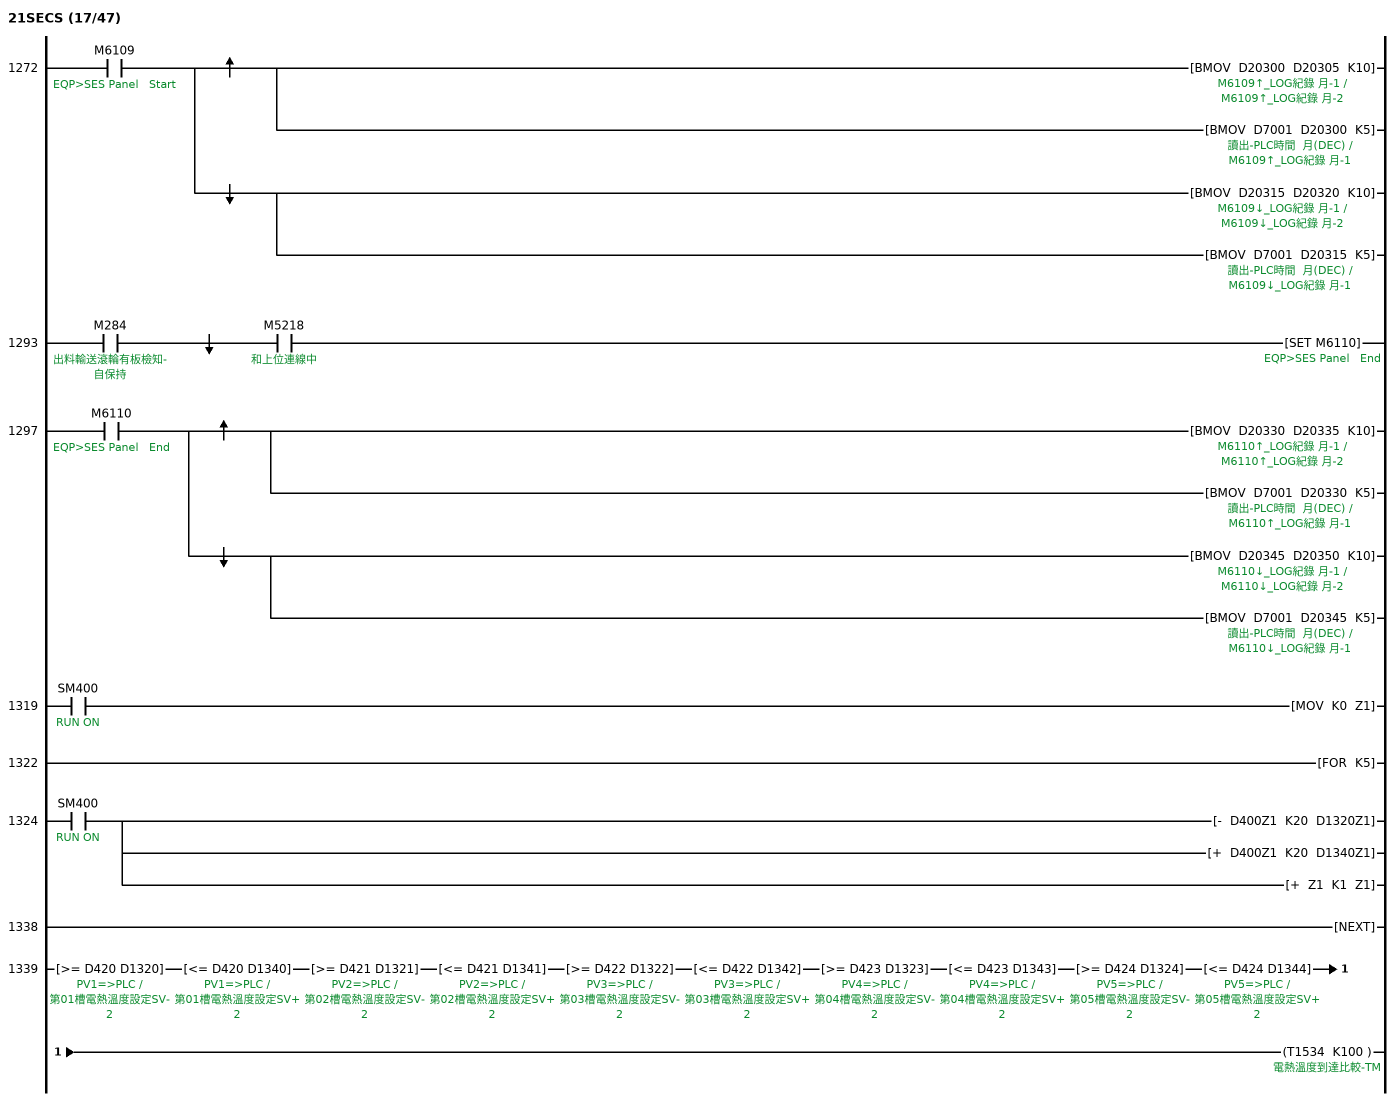
1272  LD      M6109  ; EQP>SES Panel   Start
      MPS
      MEP
      BMOV    D20300 D20305 K10  ; M6109↑_LOG紀錄 月-1 / M6109↑_LOG紀錄 月-2
      BMOV    D7001 D20300 K5
      MPP
      MEF
      BMOV    D20315 D20320 K10  ; M6109↓_LOG紀錄 月-1 / M6109↓_LOG紀錄 月-2
      BMOV    D7001 D20315 K5
1293  LD      M284  ; 出料輸送滾輪有板檢知-自保持
      MEF
      AND     M5218  ; 和上位連線中
      SET     M6110  ; EQP>SES Panel   End
1297  LD      M6110  ; EQP>SES Panel   End
      MPS
      MEP
      BMOV    D20330 D20335 K10  ; M6110↑_LOG紀錄 月-1 / M6110↑_LOG紀錄 月-2
      BMOV    D7001 D20330 K5
      MPP
      MEF
      BMOV    D20345 D20350 K10  ; M6110↓_LOG紀錄 月-1 / M6110↓_LOG紀錄 月-2
      BMOV    D7001 D20345 K5
1319  LD      SM400  ; RUN ON
      MOV     K0 Z1
1322  FOR     K5
1324  LD      SM400  ; RUN ON
      -       D400Z1 K20 D1320Z1
      +       D400Z1 K20 D1340Z1
      +       Z1 K1 Z1
1338  NEXT
1339  LD>=    D420 D1320  ; PV1=>PLC / 第01槽電熱溫度設定SV-2
      AND<=   D420 D1340  ; PV1=>PLC / 第01槽電熱溫度設定SV+2
      AND>=   D421 D1321  ; PV2=>PLC / 第02槽電熱溫度設定SV-2
      AND<=   D421 D1341  ; PV2=>PLC / 第02槽電熱溫度設定SV+2
      AND>=   D422 D1322  ; PV3=>PLC / 第03槽電熱溫度設定SV-2
      AND<=   D422 D1342  ; PV3=>PLC / 第03槽電熱溫度設定SV+2
      AND>=   D423 D1323  ; PV4=>PLC / 第04槽電熱溫度設定SV-2
      AND<=   D423 D1343  ; PV4=>PLC / 第04槽電熱溫度設定SV+2
      AND>=   D424 D1324  ; PV5=>PLC / 第05槽電熱溫度設定SV-2
      AND<=   D424 D1344  ; PV5=>PLC / 第05槽電熱溫度設定SV+2
      OUT     T1534 K100  ; 電熱溫度到達比較-TM
